{attribute 'qualified_only'}
VAR_GLOBAL
    ncAxis          : AXIS_REF;         // Link to NC axis in the I/O tree
END_VAR

(* stored: Version 1.1.0.1, ProductVersion 3.1.4026.18
   GVL GVL: Id {b9d2c063-b230-42ac-921a-7a9fce678fa7} *)
